// TIA Portal V18 export
VAR_GLOBAL   // PLC tag table "USCITE"
   Out_1 AT %Q0.0 : Bool;
   Out_2 AT %Q0.1 : Bool;
   Out_3 AT %Q0.2 : Bool;
   Out_4 AT %Q0.3 : Bool;
   Out_5 AT %Q0.4 : Bool;
   Var AT %Q0.5 : Bool;
END_VAR
